(* IEC 61131-3 sources: SIGMATEK-Jumag-Utils-Examples/delay/Class/tof, 1 file *)

(* ---- tof.st ---- *)
(*!
<Class
	Name               = "tof"
	Revision           = "0.0"
	RealtimeTask       = "false"
	CyclicTask         = "true"
	DefCyclictime      = "100 ms"
	BackgroundTask     = "false"
	Sigmatek           = "false"
	OSInterface        = "false"
	HighPriority       = "false"
	Automatic          = "false"
	UpdateMode         = "Prescan"
	SharedCommandTable = "true"
	Objectsize         = "(284,120)">
	<Channels>
		<Server Name="ClassSvr" Visualized="false" Initialize="false" WriteProtected="true" Retentive="false"/>
		<Server Name="elapsedTime" Visualized="false" Initialize="false" WriteProtected="true" Retentive="false"/>
		<Server Name="input" Visualized="false" Initialize="false" WriteProtected="false" Retentive="false"/>
		<Server Name="targetTime" Visualized="false" Initialize="true" DefValue="10000" WriteProtected="false" Retentive="false"/>
		<Server Name="timeStamp" Visualized="false" Initialize="false" WriteProtected="true" Retentive="false"/>
	</Channels>
	<Dependencies>
		<Files>
			<File Path=".\Source\delay.c"/>
		</Files>
	</Dependencies>
</Class>
*)
tof : CLASS
  //Servers:
	ClassSvr 	: SvrChCmd_DINT;
	input 	: SvrCh_DINT;
	targetTime 	: SvrCh_DINT;
	elapsedTime 	: SvrCh_UDINT;
	timeStamp 	: SvrCh_UDINT;
  //Clients:
  //Variables:
  //Functions:

	FUNCTION VIRTUAL GLOBAL CyWork
		VAR_INPUT
			EAX 	: UDINT;
		END_VAR
		VAR_OUTPUT
			state (EAX) 	: UDINT;
		END_VAR;
  //Tables:
	FUNCTION @STD
		VAR_OUTPUT
			ret_code	: CONFSTATES;
		END_VAR;
	FUNCTION GLOBAL TAB @CT_;
END_CLASS;

Function Global __cdecl DelayTof
VAR_INPUT
  IN : BOOL;
  PT : DINT;
  ET : ^UDINT;
  TIMESTAMP : ^UDINT;
  CLOCK : UDINT;
END_VAR
VAR_OUTPUT
  Q : BOOL;
END_VAR;

FUNCTION VIRTUAL GLOBAL tof::CyWork
	VAR_INPUT
		EAX 	: UDINT;
	END_VAR
	VAR_OUTPUT
		state (EAX) 	: UDINT;
	END_VAR
  VAR
  	x : BOOL;
  END_VAR

  if (input = 1)  then
    x := true;
    else
      x := false;
  end_if;

  ClassSvr := DelayTof(IN:=x, PT:=targetTime, ET:=#elapsedTime, TIMESTAMP:=#timestamp, CLOCK:=ops.tAbsolute);

	state := READY;

END_FUNCTION
